FUNCTION_BLOCK INTERNAL FB_Winter EXTENDS FB_SeasonBase
VAR
END_VAR

METHOD ChangeToWinterTyres
VAR_INPUT
END_VAR
THIS^._nTyresType := 0;
Tc2_System.ADSLOGSTR(msgCtrlMask := THIS^._nLogLevel,
                     msgFmtStr := 'Changed to winter tyres',
                     strArg := '');
END_METHOD

METHOD FB_init : BOOL
VAR_INPUT
    bInitRetains:           BOOL; // if TRUE, the retain variables are initialized (warm start / cold start)
    bInCopyCode:            BOOL;  // if TRUE, the instance afterwards gets moved into the copy code (online change)
    ipStateMachine:         I_StateMachine;
    ipParentObject:         I_Object;
END_VAR
THIS^._eState := E_Season.Winter;
END_METHOD

METHOD  NextSeason
VAR_INPUT
END_VAR
THIS^.ipStateMachine.SetState(THIS^.ipSeasonCtrl.StateSpring);
END_METHOD

METHOD OnEntry
VAR_INPUT
END_VAR
SUPER^.OnEntry();
THIS^._bWindBlowing     := FALSE;
THIS^._bRaining         := FALSE;
THIS^._bSunShining      := FALSE;
THIS^._bSnowing         := TRUE;
THIS^._nLeavesState     := 0;
END_METHOD

END_FUNCTION_BLOCK

(* stored: Version 1.1.0.1, ProductVersion 3.1.4024.12
   POU FB_Winter: Id {880ccb34-50d9-0359-2ea3-2a8967823e9a}, SpecialFunc None
   Method ChangeToWinterTyres: Id {903cf646-55f0-0fd1-2691-f4f4f71902d2}
   Method FB_init: Id {94d78c1b-eb3a-0116-069f-896cca73648e}
   Method NextSeason: Id {57d885c3-6074-007f-1b9c-f8ed74bb1904}
   Method OnEntry: Id {4eccdcb9-6ff6-0a8d-1f07-e7f075928458} *)
